{attribute 'qualified_only'}
{attribute 'strict'}
TYPE E_LAMP_SUBSTATE :
(
	NONE				:= 0,
	
	NOTOP_NOTREADY		:= 100,
	NOTOP_INITIALIZING	:= 102,
	NOTOP_READY_OFF		:= 103,
	NOTOP_READY_ON		:= 104,
	NOTOP_ERROR			:= 199,
	
	OP_DISABLING		:= 205,
	OP_OFF				:= 206,            
	OP_SWITCHING_OFF	:= 207,           
	OP_COOLING			:= 208,
	OP_ON				:= 209,
	OP_SWITCHING_ON		:= 210,
	OP_WARMING			:= 211,
	OP_ERROR			:= 299
);
END_TYPE

(* stored: Version 1.1.0.1, ProductVersion 3.1.4022.16
   DUT E_LAMP_SUBSTATE: Id {799404c9-da36-48d5-9ce1-118394e18490} *)
